FUNCTION_BLOCK ModbusMaster (* Modbus Master *)
  (* Standard: 61499-2; Description: Copyright (c) 2024 Martin Erich Jobst This program and the accompanying materials are made available under the terms of the Eclipse Public License 2.0 which is available at https://www.eclipse.org/legal/epl-2.0/ SPDX-License-Identifier: EPL-2.0 *)
  (* Version 1.0, 2024-09-12, Martin Erich Jobst *)
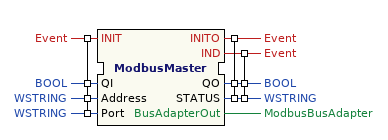
  EVENT_INPUT
    INIT WITH QI, Address, Port; (* Service Initialization *)
  END_EVENT
  EVENT_OUTPUT
    INITO WITH QO, STATUS; (* Initialization Confirm *)
    IND WITH QO, STATUS; (* Indication from Resource *)
  END_EVENT
  VAR_INPUT
    QI : BOOL; (* Event Input Qualifier *)
    Address : WSTRING; (* Modbus Address *)
    Port : WSTRING; (* Modbus Port *)
  END_VAR
  VAR_OUTPUT
    QO : BOOL; (* Event Output Qualifier *)
    STATUS : WSTRING; (* Service Status *)
  END_VAR
  PLUGS
    BusAdapterOut : ModbusBusAdapter;
  END_PLUGS
END_FUNCTION_BLOCK
